FUNCTION SCODE_CODE : DWORD
(* Helper function: returns the lower word of error code *)
VAR_INPUT
	sc		: DWORD;
END_VAR

SCODE_CODE := 16#FFFF AND sc;

END_FUNCTION

(* stored: Version 1.1.0.1, ProductVersion 3.1.0.19
   POU SCODE_CODE: Id {22f2198f-6d3d-4db8-96d9-e383780179d6} *)
